SYSTEM FLASHER_TEST (* Flasher Test System Configuration *)
  (* Standard: 61499-1 *)
  (* Version 0.4, 2007-11-07, JHC, Holobloc Inc, Changed RUNSTOP to RADIO_BOOL+E_SWITCH. *)
  (* Version 0.3, 2006-10-26, JHC, Holobloc Inc, Adapted to new FLASHER4 without INITO. *)
  (* Version 0.2, 2006-10-25, JHC, Holobloc Inc, Moved to doc folder. *)
  (* Version 0.1, 2001-07-31, JHC, Rockwell Automation, Changed IN_TIME to IN_ANY, adjusted height. *)
  (* Version 0.0, 2001-02-22, JHC, Rockwell Automation *)
  DEVICE FLASHER : FRAME_DEVICE(BOUNDS := [100,100,350,100], GRID := [1,1])
    RESOURCE RES1 : PANEL_RESOURCE
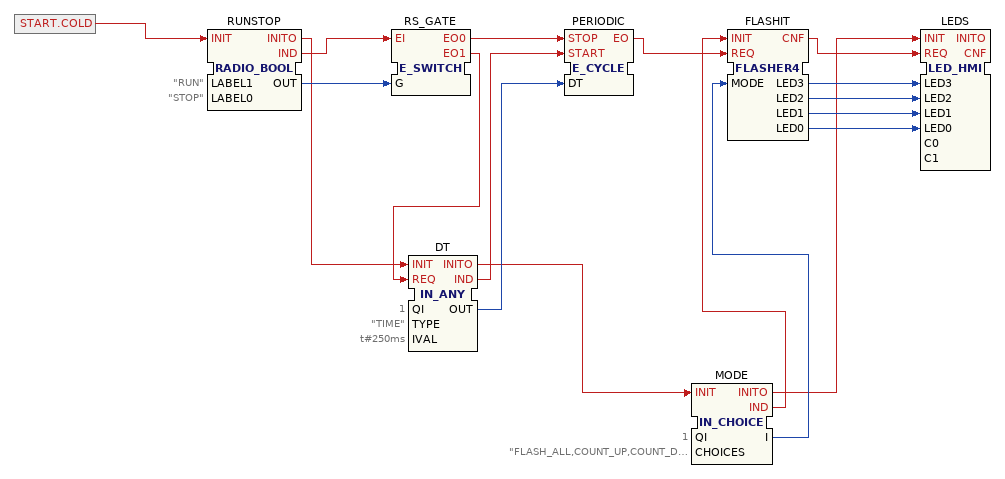
      FBS
        DT : IN_ANY(QI := 1, TYPE := "TIME", IVAL := t#250ms);
        PERIODIC : E_CYCLE;
        MODE : IN_CHOICE(QI := 1, CHOICES := "FLASH_ALL,COUNT_UP,COUNT_DOWN,CHASE_UP,CHASE_DOWN");
        FLASHIT : FLASHER4;
        LEDS : LED_HMI;
        RUNSTOP : RADIO_BOOL(LABEL1 := "RUN", LABEL0 := "STOP");
        RS_GATE : E_SWITCH;
      END_FBS
      EVENT_CONNECTIONS
        DT.INITO TO MODE.INIT;
        MODE.INITO TO LEDS.INIT;
        MODE.IND TO FLASHIT.INIT;
        PERIODIC.EO TO FLASHIT.REQ;
        FLASHIT.CNF TO LEDS.REQ;
        START.COLD TO RUNSTOP.INIT;
        RUNSTOP.INITO TO DT.INIT;
        RUNSTOP.IND TO RS_GATE.EI;
        RS_GATE.EO0 TO PERIODIC.STOP;
        RS_GATE.EO1 TO DT.REQ;
        DT.IND TO PERIODIC.START;
      END_CONNECTIONS
      DATA_CONNECTIONS
        DT.OUT TO PERIODIC.DT;
        MODE.I TO FLASHIT.MODE;
        FLASHIT.LED3 TO LEDS.LED3;
        FLASHIT.LED2 TO LEDS.LED2;
        FLASHIT.LED1 TO LEDS.LED1;
        FLASHIT.LED0 TO LEDS.LED0;
        RUNSTOP.OUT TO RS_GATE.G;
      END_CONNECTIONS
    END_RESOURCE
  END_DEVICE
END_SYSTEM
